TYPE ST_GSR_6_1 :
(**************************************************************************************
 * 	Application		:	BoxControl Framework
 *	Revision		:	$Revision: 404529 $
 *	Revision date	:	$Date: 2018-04-23 08:21:38 +0200 (Mo., 23 Apr 2018) $
 *	Last changed by	:	$Author: b7bolm $
 *	URL				:	$URL: http://almscdc.swisslog.com/repo/SWPD/Development/BoxControlFramework/20_Release/trunk/01_Software/BCF/BCF/JumpStart/20_Product/10_App/11_Com/10_Lib/10_Conv/12_MFCS/11_SIS/01_DUTs/11_SIS_6_1/ST_GSR_6_1.TcDUT $
 *
 *	Purpose			:	GCR Structure
 *
 * ------------------------------------------------------------------------------------
 *	Copyright Swisslog [IP AG], Switzerland. All rights reserved.
 * 
 * ------------------------------------------------------------------------------------
 *	
 * 	Revision History: 
 *
 * 	VERSION			DATE			INITIALS			DESCRIPTION
 *	0.1				01.01.2001		swl					Example
 *
 **************************************************************************************)
STRUCT
	GroupName		: STRING(SIS_6_1.POSITION_STRINGLENGTH); // 12 Digit SIS Group Name MM-GGG-0000-000 
	Mode			: STRING(SIS_6_1.MODE_STRINGLENGTH); // 1 Digit Mode 
	State			: STRING(SIS_6_1.STATE_STRINGLENGTH); // 1 Digit State 
	ErrorState		: STRING(SIS_6_1.ERRORSTATE_STRINGLENGTH); // 1 Digit error State 
	ErrorCode		: STRING(SIS_6_1.ERRORCODE_STRINGLENGTH); // 4 Digit Return Code 
	ErrorType		: STRING(SIS_6_1.ERRORTYPE_STRINGLENGTH); // 1 Digit Error Type 
	ErrorInformation: STRING(SIS_6_1.ERRORINFORMATION_STRINGLENGTH); // 5 Chars Error Information 
	Variable		: STRING(SIS_6_1.CONTROLVARIABLE_STRINGLENGTH); // 4 DigitControl code variable 
	ReturnCode		: STRING(SIS_6_1.ERRORCODE_STRINGLENGTH); // 4 Digit return code
END_STRUCT
END_TYPE

(* stored: Version 1.1.0.1, ProductVersion 3.1.4022.12
   DUT ST_GSR_6_1: Id {9b67531b-3a97-45d3-8419-f01240aaf766} *)
